// TIA Portal V20 export
DATA_BLOCK "Config"   // DB198
// stored: MemoryReserve 100, Namespace Unit1.Em3
   VAR
      em : "LAF_typeEmConfiguration";   // Configuration of EM Parameters
      axis : Array[1.._.U1EM3_NO_OF_AXES] of DB_ANY;
   END_VAR
   VAR RETAIN
      cmMasterVirtualAxis : "LBC_typeAxisControlConfiguration";
      cmUnwinderVirtualAxis : "LBC_typeAxisControlConfiguration";
      cmDancerRegulatorOnOff : "LBC_typeTwoWayActuatorConfiguration";
      cmDancerSafetyPinIdlePosition : "LBC_typeDigitalSignalConfiguration";
      cmLoadCellAnalogInput : "LBC_typeAnalogInputConfiguration";
      cmDancerEncoderAnalogInput : "LBC_typeAnalogInputConfiguration";
      cmDancerElectroPneumaticRegulatorAnalogOutput : "LBC_typeAnalogOutputConfiguration";
      cmWebGuideEpc : "LER_typeCON600Configuration";
   END_VAR
BEGIN
END_DATA_BLOCK
